{attribute 'hide_all_locals'}
PROGRAM EthercatHelper
VAR
	fbReadDeviceName	: Tc2_IoFunctions.IOF_GetBoxNameByAddr;
	nMasterId			: UDINT;
	fbCoe				: FB_CoeReadWrite;
END_VAR

METHOD CoE : REFERENCE TO FB_CoeReadWrite
VAR_INPUT
END_VAR
CoE REF= fbCoE;
END_METHOD

METHOD PUBLIC GetBoxNameByAddress : T_MaxString
VAR_INPUT
	PlcRuntimeNetId		: Tc2_System.T_AmsNetID; // NetId of the PLC where the devuce is located
	AmsNetId			: AMSADDR; // NetId of the box
	outError			: REFERENCE TO BOOL;	// If an error occurs while executing, method will provide the error flag here. This is a pointer to YOUR boolean error variable.
END_VAR

VAR
	sNetId	: Tc2_System.T_AmsNetID;
END_VAR
sNetId := AdsHelper.NetIdToString(AmsNetId.netId);
fbReadDeviceName(
	NETID := PlcRuntimeNetId,
	DEVICEID := AdsHelper.GetEthercatMasterIdFromNetIdString(netId := sNetId),
	BOXADDR := AmsNetId.port,
	START := NOT fbReadDeviceName.BUSY);
	
outError := fbReadDeviceName.ERR;
GetBoxNameByAddress := fbReadDeviceName.BOXNAME;
END_METHOD

END_PROGRAM

(* stored: Version 1.1.0.1, ProductVersion 3.1.4024.13
   POU EthercatHelper: Id {18c8e82e-8363-065e-3a67-80a80ad75944}, SpecialFunc None
   Method CoE: Id {64b56a36-5c04-024e-00fa-396319932b60}
   Method GetBoxNameByAddress: Id {05a15158-8102-075e-26df-9833faf2f947} *)
